// Mitsubishi GX Works2 project: test   PLC: Q06H

PROGRAM MAIN
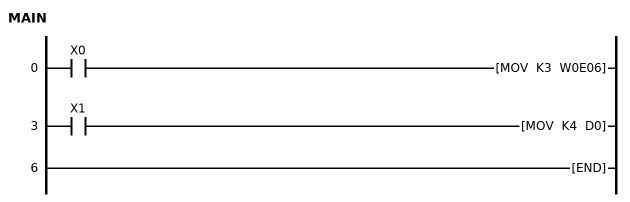
0     LD      X0
      MOV     K3 W0E06
3     LD      X1
      MOV     K4 D0
6     END
END_PROGRAM
